// TIA Portal V16 export
// export: Created 2021-09-08T12:46:15.6972977Z, ExportSetting WithDefaults, DisplayName Totally Integrated Automation Portal, DisplayVersion V16 Update 3, DisplayName TIA Portal Version Control Interface, DisplayVersion V16 Update 2, DisplayName TIA Portal Openness, DisplayVersion V16 Update 3, DisplayName TIA Portal Teamcenter Gateway, DisplayVersion V16, DisplayName STEP 7 Professional, DisplayVersion V16 Update 3, DisplayName STEP 7 Safety, DisplayVersion V16, DisplayName WinCC Advanced, DisplayVersion V16 Update 3
TYPE "Ai"
// stored: IsFailsafeCompliant false
   STRUCT
      emMax_En { ExternalAccessible := 'False'; ExternalVisible := 'False'; ExternalWritable := 'False'; S7_SetPoint := 'True'} : Bool;   // Аварийный верхний 1-проверять
      emMin_En { ExternalAccessible := 'False'; ExternalVisible := 'False'; ExternalWritable := 'False'; S7_SetPoint := 'True'} : Bool;   // Аварийный нижний 1-проверять
      wrnMax_En { ExternalAccessible := 'False'; ExternalVisible := 'False'; ExternalWritable := 'False'; S7_SetPoint := 'True'} : Bool;   // Предупредительный верхний 1-проверять
      wrnMin_En { ExternalAccessible := 'False'; ExternalVisible := 'False'; ExternalWritable := 'False'; S7_SetPoint := 'True'} : Bool;   // Предупредительный нижний 1-проверять
      curEmMax { ExternalAccessible := 'False'; ExternalVisible := 'False'; ExternalWritable := 'False'} : Bool;   // В данный момент значение выше аварийного максимума
      curEmMin { ExternalAccessible := 'False'; ExternalVisible := 'False'; ExternalWritable := 'False'} : Bool;   // В данный момент значение ниже аварийного минимума
      curWnMax { ExternalAccessible := 'False'; ExternalVisible := 'False'; ExternalWritable := 'False'} : Bool;   // В данный момент значение выше предупредительного максимума
      curWnMin { ExternalAccessible := 'False'; ExternalVisible := 'False'; ExternalWritable := 'False'} : Bool;   // В данный момент значение ниже предупредительного минимума
      emMax { ExternalAccessible := 'False'; ExternalVisible := 'False'; ExternalWritable := 'False'} : Bool;   // Сработала сигнализация - аварийный максимум
      emMin { ExternalAccessible := 'False'; ExternalVisible := 'False'; ExternalWritable := 'False'} : Bool;   // Сработала сигнализация - аварийный минимум
      wnMax { ExternalAccessible := 'False'; ExternalVisible := 'False'; ExternalWritable := 'False'} : Bool;   // Сработала сигнализация - предупредительный максимум
      wnMin { ExternalAccessible := 'False'; ExternalVisible := 'False'; ExternalWritable := 'False'} : Bool;   // Сработала сигнализация - предупредительный минимум
      Err : Bool;   // Наличие ошибок канала / Налицие ошибок канала
      badParam { ExternalVisible := 'False'} : Bool;   // Неправильные параметры
      overFlow { ExternalVisible := 'False'} : Bool;   // Перегрузка канала
      wireBreak { ExternalVisible := 'False'} : Bool;   // Обрыв провода
      SimEnable { S7_SetPoint := 'True'} : Bool;   // Включение симуляции
      disableParLessZero { S7_SetPoint := 'True'} : Bool := 1;   // 1-Запрет значений меньше нуля, типа плавающих значений
      modeAck { S7_SetPoint := 'True'} : Bool := 1;   // 1-сброс по общему сбросу аварий, 0-сброс после исчезновения условия
      ackAll : Bool;   // сброс всех событий
      ack { ExternalVisible := 'False'} : Byte;   // Байт сброса ошибок
      State : Word;   // Код качества
      Par_code { ExternalVisible := 'False'} : Int;   // Код канала
      Par : Real;   // Значение параметра в технологических единицах
      rngUpLm { ExternalVisible := 'False'; S7_SetPoint := 'True'} : Real := 200.0;   // Максимум диапазона измерения
      rngLwLm { ExternalVisible := 'False'; S7_SetPoint := 'True'} : Real;   // Минимум диапазона измерения
      emrMax { ExternalVisible := 'False'; S7_SetPoint := 'True'} : Real := 190.0;   // Технологический верхний аварийный предел
      emrMaxTime { ExternalVisible := 'False'; S7_SetPoint := 'True'} : Real := 5.0;   // Время задержки для срабатывания аварии по Аварийному верхнему пределу
      emrMin { ExternalVisible := 'False'; S7_SetPoint := 'True'} : Real := 10.0;   // Технологический нижний аварийный предел
      emrMinTime { ExternalVisible := 'False'; S7_SetPoint := 'True'} : Real := 5.0;   // Время задержки для срабатывания аварии по Аварийному нижниму пределу
      wrnMax { ExternalVisible := 'False'; S7_SetPoint := 'True'} : Real := 150.0;   // Технологический верхний предупредительный предел
      wrnMaxTime { ExternalVisible := 'False'; S7_SetPoint := 'True'} : Real := 5.0;   // Время задержки для срабатывания аварии по Предупредительному верхнему пределу
      wrnMin { ExternalVisible := 'False'; S7_SetPoint := 'True'} : Real := 20.0;   // Технологический нижний предупредительный предел
      wrnMinTime { ExternalVisible := 'False'; S7_SetPoint := 'True'} : Real := 5.0;   // Время задержки для срабатывания аварии по Предупредительному нижниму пределу
      Par_mA { ExternalVisible := 'False'} : Real;   // Значение параметра в мА
      SimValue { ExternalVisible := 'False'} : Real;   // Значение симуляции
      curTimeEmrMin { ExternalAccessible := 'False'; ExternalVisible := 'False'; ExternalWritable := 'False'} : Real;   // Текуще значение таймера
      curTimeWrnMin { ExternalAccessible := 'False'; ExternalVisible := 'False'; ExternalWritable := 'False'} : Real;   // Текуще значение таймера
      curTimeWrnMax { ExternalAccessible := 'False'; ExternalVisible := 'False'; ExternalWritable := 'False'} : Real;   // Текуще значение таймера
      curTimeEmrMax { ExternalAccessible := 'False'; ExternalVisible := 'False'; ExternalWritable := 'False'} : Real;   // Текуще значение таймера
      Spare_0 { ExternalAccessible := 'False'; ExternalVisible := 'False'; ExternalWritable := 'False'} : Word;
      Spare_1 { ExternalAccessible := 'False'; ExternalVisible := 'False'; ExternalWritable := 'False'} : Word;
      Spare_2 { ExternalAccessible := 'False'; ExternalVisible := 'False'; ExternalWritable := 'False'} : Word;
      Spare_3 { ExternalAccessible := 'False'; ExternalVisible := 'False'; ExternalWritable := 'False'} : Word;
      Spare_4 { ExternalAccessible := 'False'; ExternalVisible := 'False'; ExternalWritable := 'False'} : Word;
      Spare_5 { ExternalAccessible := 'False'; ExternalVisible := 'False'; ExternalWritable := 'False'} : Word;
      Spare_6 { ExternalAccessible := 'False'; ExternalVisible := 'False'; ExternalWritable := 'False'} : Word;
      Spare_7 { ExternalAccessible := 'False'; ExternalVisible := 'False'; ExternalWritable := 'False'} : Word;
      Spare_8 { ExternalAccessible := 'False'; ExternalVisible := 'False'; ExternalWritable := 'False'} : Word;
      Spare_9 { ExternalAccessible := 'False'; ExternalVisible := 'False'; ExternalWritable := 'False'} : Word;
      Spare_10 { ExternalAccessible := 'False'; ExternalVisible := 'False'; ExternalWritable := 'False'} : Word;
      Spare_11 { ExternalAccessible := 'False'; ExternalVisible := 'False'; ExternalWritable := 'False'} : Word;
   END_STRUCT;
END_TYPE
